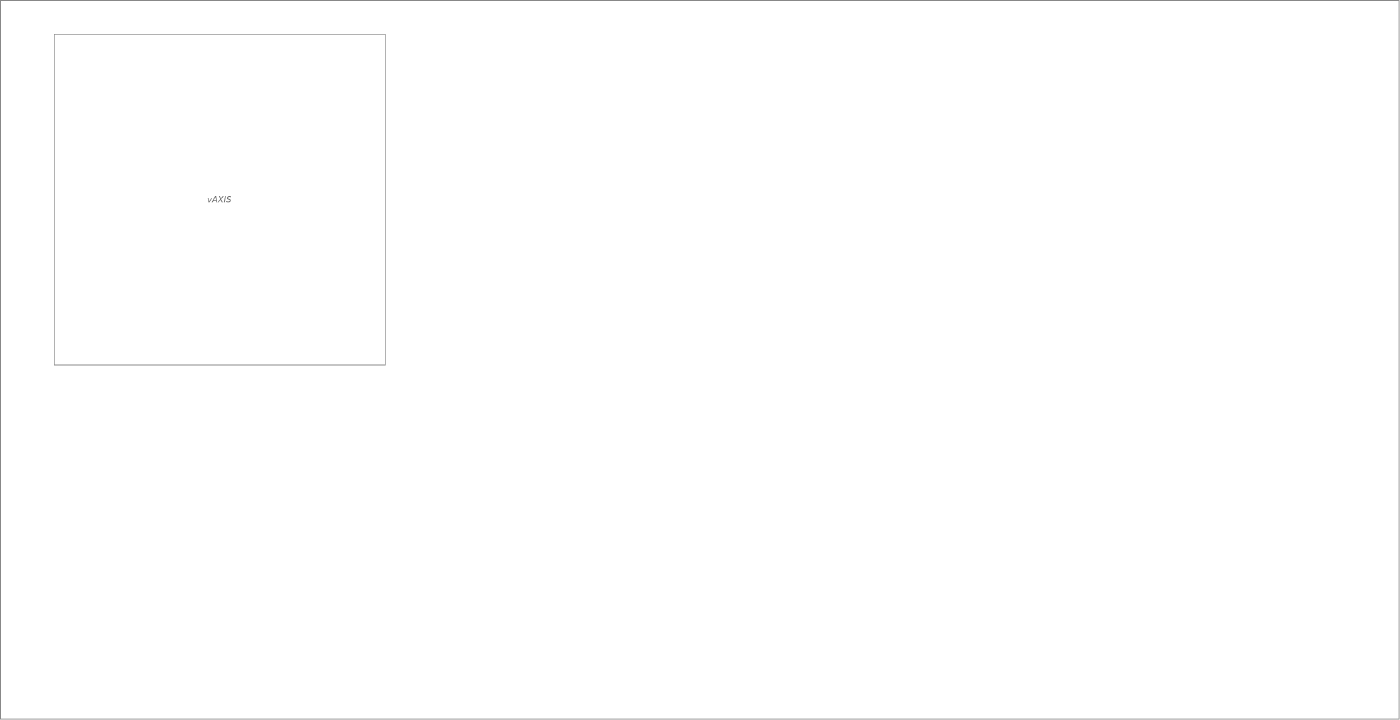
VISUALIZATION AXES_SCREEN  // 1690x870
    Frame (65,41 400x400)
        shows vAXIS(vAxis := MAIN_CONV)
END_VISUALIZATION

(* stored: Version 1.1.0.1, ProductVersion 3.1.4024.12
   Visu AXES_SCREEN: Id {dc606aed-ddbd-4585-acdd-725e8541e359} *)
